(* Logix 5000 project; controller Kinematics_Delta_5D_with_Pick_n_Place 1756-L85E rev 33.11; software revision 33.00 *)

TASK MainTask (continuous, watchdog 500 ms) : MainProgram
TASK MotionEventTask (task) : VectorDynamics

MODULES
   Local : 1756-L85E (ICP 0, rev 33.11)
END_MODULES

TYPE SimOutputs :
STRUCT
   NumValues : DINT;   // Count of variables in the image
   D5_800_Y_ACT : REAL;   // Physics://physics/physics/D5-800/D5-800?_Y_ACT
   D5_800_Z_ACT : REAL;   // Physics://physics/physics/D5-800/D5-800?_Z_ACT
   D5_800_X_ACT : REAL;   // Physics://physics/physics/D5-800/D5-800?_X_ACT
   D5_800_R1_ACT : REAL;   // Physics://physics/physics/D5-800/D5-800?_R1_ACT
   D5_800_R2_ACT : REAL;   // Physics://physics/physics/D5-800/D5-800?_R2_ACT
   D5_800_GRIP : BOOL;   // Physics://physics/physics/D5-800/D5-800?_GRIP
END_STRUCT
END_TYPE

ADD_ON_INSTRUCTION deltaHomeArms   (* revision 1.0 *)

ROUTINE EnableInFalse   (* ladder *)
END_ROUTINE

ROUTINE Logic   (* ladder *)
END_ROUTINE
END_ADD_ON_INSTRUCTION

ADD_ON_INSTRUCTION Forward_Kinematics   (* revision 1.0, vendor Rockwell Automation *)
// This AOI will perform forward kinematics for Six axis articulated independent robot

ROUTINE Logic   (* structured text *)
   
END_ROUTINE
END_ADD_ON_INSTRUCTION

ADD_ON_INSTRUCTION homeToPositionError   (* revision 1.0, ExecuteEnableInFalse *)

ROUTINE EnableInFalse   (* ladder *)
END_ROUTINE

ROUTINE Logic   (* ladder *)
END_ROUTINE
END_ADD_ON_INSTRUCTION

ADD_ON_INSTRUCTION PICKPLACE   (* revision 1.0, ExecutePrescan *)
// Revision note:
// This AOI exhibits the PICK and PLACE behavior for a virtual cartesian axes.

ROUTINE Logic   (* ladder *)
END_ROUTINE

ROUTINE Prescan   (* ladder *)
// Move Step
END_ROUTINE
END_ADD_ON_INSTRUCTION

VAR_GLOBAL   (* controller tags *)
   a1_move_to_initialposition : BOOL;
   a2_mctTurnOn : BOOL;
   AccDec : REAL := 6666.665;
   Actual_Position_axis : REAL[3] := ([0] := 281.0, [2] := -1065.0219);
   AutoBrake : BOOL;
   Axis_Homing : BOOL;
   backOffAngle : REAL := 30.0;
   brakeAutoConstant : SINT; {constant}
   brakeReleaseConstant : SINT := 1; {constant}
   Cart_Vector_Speed_Sqr : REAL;
   Cart_Vector_Velocity_Sqr : REAL;
   CartSpeed : REAL := 500.0;
   CartVectorVelocity : REAL;
   CommandTolerance : REAL := 50.0;
   Counter : COUNTER := (PRE := 2, ACC := 1);
   CS_XYZRxRyRz : COORDINATE_SYSTEM;
   CycleTime : TIMER := (PRE := 99999, ACC := 99999, EN := 1, DN := 1);
   Delta5D_J1J2J3J4J5 : COORDINATE_SYSTEM;
   DeltaHomeArms : BOOL;
   DHA : deltaHomeArms;
   DownDist : REAL[3] := ([2] := -60.0);
   Downdistance : REAL := 80.0;
   DownDistBack : REAL := -120.0;
   dyn_data : DYNAMICS_DATA := (TimeUnits := 1, Profile := 1, Speed := 10.0, Acceleration := 5.0, Deceleration := 5.0, AccelerationJerk := 100.0, DecelerationJerk := 100.0, OrientationSpeed := 10.0, OrientationAcceleration := 30.0, OrientationDeceleration := 30.0);
   forAllAxes : BOOL;
   forArmsOnly : BOOL;
   forAxis1 : BOOL := 1;
   forAxis2 : BOOL := 1;
   forAxis3 : BOOL := 1;
   forAxis4 : BOOL;
   forAxis5 : BOOL;
   forNoAxes : BOOL;
   H2PE_1 : homeToPositionError;
   HalfHorizonMCLM : MOTION_INSTRUCTION := (FLAGS := -1442840576, EN := 1, DN := 1, PC := 1);
   homeMCPM : PATH_DATA[1] := ([0].InterpolationType := 1, [0].Position[0] := -20.012327, [0].Position[1] := 79.85217, [0].Position[2] := -7.858248, [0].Position[3] := -0.007234964, [0].Position[4] := 18.006336, [0].Position[5] := -20.005451, [0].RobotConfiguration := 6, [0].TerminationType := 1);
   HomePos : REAL[8] := ([0] := -20.012327, [1] := 79.85217, [2] := -7.858248, [3] := -0.007234964, [4] := 18.006336, [5] := -20.005451);
   HomeToTorque : BOOL;
   HorizDistance : REAL[3] := ([0] := -150.0);
   HorizDistBack : REAL := -360.0;
   HorizontalDistance : REAL := 360.0;
   InitialMclm1 : MOTION_INSTRUCTION;
   InitialPos : BOOL;
   Initiate_MCTO : BOOL;
   J1_Pos : REAL := 28.4;
   J1_v : AXIS_VIRTUAL;
   J2_Pos : REAL := 4.911;
   J2_v : AXIS_VIRTUAL;
   J3_Pos : REAL := -0.165;
   J3_v : AXIS_VIRTUAL;
   J4_Pos : REAL := -36.107;
   J4_v : AXIS_VIRTUAL;
   j4Angle : REAL := 180.0;
   j4AngleReturn : REAL := -180.0;
   J5_Pos : REAL := 35.032;
   J5_v : AXIS_VIRTUAL;
   j5Angle : REAL := 120.0;
   j5AngleReturn : REAL := -120.0;
   J6_Pos : REAL := -78.86052;
   J6_v : AXIS_VIRTUAL;
   junk1 : BOOL;
   LocalStep : DINT;
   LocalStep1 : DINT := 3;
   mah1 : MOTION_INSTRUCTION := (FLAGS := 704643072, DN := 1, PC := 1, STATE := 17);
   mah2 : MOTION_INSTRUCTION := (FLAGS := 704643072, DN := 1, PC := 1, STATE := 17);
   mah3 : MOTION_INSTRUCTION := (FLAGS := 704643072, DN := 1, PC := 1, STATE := 17);
   mah4 : MOTION_INSTRUCTION := (FLAGS := 704643072, DN := 1, PC := 1, STATE := 17);
   mah5 : MOTION_INSTRUCTION := (FLAGS := 704643072, DN := 1, PC := 1, STATE := 17);
   Mah_Ctr : MOTION_INSTRUCTION[10] := ([0].FLAGS := 33554432, [1].FLAGS := 33554432, [2].FLAGS := 33554432, [3].FLAGS := 33554432, [4].FLAGS := 33554432);
   maj1 : MOTION_INSTRUCTION := (FLAGS := 637534208, DN := 1, IP := 1);
   majMaster : REAL := 1.0;
   MAM_TO_ZERO : MOTION_INSTRUCTION[3] := ([0].FLAGS := 33554432, [1].FLAGS := 33554432, [2].FLAGS := 33554432);
   MAS : MOTION_INSTRUCTION[5] := ([0].FLAGS := 33554432, [1].FLAGS := 33554432, [2].FLAGS := 33554432, [3].FLAGS := 33554432, [4].FLAGS := 33554432);
   mas1 : MOTION_INSTRUCTION := (FLAGS := 33554432);
   masterZeroAngle : REAL := -82.04;
   MaxAccDec : REAL;
   MaxAccel : REAL := 70000.0;
   mccd1 : MOTION_INSTRUCTION;
   mccdOn : BOOL;
   mcpm : MOTION_INSTRUCTION[10] := ([0].FLAGS := 33554432, [1].FLAGS := 33554432, [2].FLAGS := 33554432, [3].FLAGS := 33554432, [4].FLAGS := 33554432, [5].FLAGS := 33554432, [6].FLAGS := 33554432, [7].FLAGS := 33554432, [8].FLAGS := 33554432);
   MCPM_Absolute_Move : BOOL;
   mcpm_ctr : MOTION_INSTRUCTION := (FLAGS := 33554432);
   MCPM_Incremental_Move : BOOL;
   mcpm_path : PATH_DATA[10] := ([0].InterpolationType := 1, [0].Position[0] := 100.0, [0].Position[1] := 200.0, [0].Position[2] := 300.0, [0].Position[3] := 30.0, [0].Position[4] := 20.0, [0].Position[5] := 10.0, [0].TerminationType := 1, [1].InterpolationType := 1, [1].Position[0] := 200.0, [1].Position[1] := 300.0, [1].Position[2] := 100.0, [1].Position[3] := 20.0, [1].Position[4] := 30.0, [1].Position[5] := 10.0, [1].TerminationType := 1, [2].InterpolationType := 1, [2].TerminationType := 1, [3].InterpolationType := 1, [3].Position[0] := 400.0, [3].Position[1] := 250.0, [3].Position[2] := 350.0, [3].Position[3] := 60.0, [3].Position[4] := 45.0, [3].Position[5] := 65.0);
   MCPM_RzMove_Coupling : BOOL;
   MCPM_with_WorkTool : BOOL;
   MCSOn : BOOL;
   mct1 : MOTION_INSTRUCTION := (FLAGS := 33554432);
   mctOn : BOOL := 1;
   mdcc1 : MOTION_INSTRUCTION := (FLAGS := 33554432);
   MotionAxisHome : BOOL;
   MotionAxisStop : BOOL;
   MotionServoOff : BOOL;
   MotionServoOn : BOOL;
   MoveArmsToZero : BOOL;
   MoveDown : BOOL;
   moveSpeed : REAL := 2.0;
   moveToZeroAccelAndJerk : REAL := 50.0;
   moveToZeroSpeed : REAL := 5.0;
   MSF : MOTION_INSTRUCTION[5] := ([0].FLAGS := 33554432, [1].FLAGS := 33554432, [2].FLAGS := 33554432, [3].FLAGS := 33554432, [4].FLAGS := 33554432);
   MSO : MOTION_INSTRUCTION[5] := ([0].FLAGS := 33554432, [1].FLAGS := 33554432, [2].FLAGS := 33554432, [3].FLAGS := 33554432, [4].FLAGS := 33554432);
   msoJ1 : MOTION_INSTRUCTION := (FLAGS := 33554432);
   msoJ2 : MOTION_INSTRUCTION := (FLAGS := 33554432);
   msoJ3 : MOTION_INSTRUCTION := (FLAGS := 33554432);
   msoJ4 : MOTION_INSTRUCTION := (FLAGS := 33554432);
   msoJ5 : MOTION_INSTRUCTION := (FLAGS := 33554432);
   OldCartSpeed : REAL;
   Ori_Vector_Speed_Sqr : REAL;
   Ori_Vector_Velocity_Sqr : REAL;
   ort : REAL[3];
   OrtVectorVelocity : REAL;
   path : PATH_DATA[10];
   PathPositions : REAL[8] := ([0] := 476.104, [1] := 2.682, [2] := -1200.037, [3] := 180.0);
   PathPositions1 : REAL[8] := ([0] := 498.811, [1] := -51.046, [2] := -885.044, [4] := -90.0, [5] := 135.0);
   PathPositions2 : REAL[8] := ([0] := -48.009, [1] := -19.226, [2] := -930.044, [3] := 180.0, [5] := -45.0);
   PathPositions3 : REAL[8] := ([0] := -145.893, [1] := 2.719, [2] := -1155.048, [4] := -90.0);
   PathPositions4 : REAL[8] := ([0] := 400.00003, [1] := 199.99995, [2] := 300.0, [3] := -179.99901, [4] := -0.0009865595, [5] := 90.0);
   PathPositions5 : REAL[8] := ([0] := 399.99997, [1] := -145.68004, [2] := 300.0, [3] := -179.999, [4] := -0.0010051423, [5] := 180.0);
   PathPositions6 : REAL[8] := ([0] := 399.99597, [1] := -145.68709, [2] := 7.3754336e-10, [3] := -179.99799, [4] := -0.0010051426, [5] := 180.0);
   pauseMove : DINT := 1;
   Pick_cycles_per_minute : REAL := 0.6000059;
   PickPlace2 : PICKPLACE;
   Place : BOOL;
   posArray : REAL[3] := ([0] := -180.0, [2] := -620.0);
   posErrThresh : REAL := 0.4;
   ReleaseBrake : BOOL;
   Robot : MOTION_GROUP;
   Rx : AXIS_VIRTUAL;
   Ry : AXIS_VIRTUAL;
   Rz : AXIS_VIRTUAL;
   simOutputs : SimOutputs := (NumValues := 6, D5_800_Z_ACT := -0.74696803, D5_800_X_ACT := 0.25423348, D5_800_R1_ACT := 1.2645825);
   SpeedOverwrite : BOOL;
   Start_AOI : BOOL;
   Start_MCPM : BOOL;
   Start_PickPlace : BOOL;
   step : DINT;
   Stop_Program : BOOL;
   T_CycleFrequency : REAL := 0.6000059;
   TermType1 : DINT := 1;
   test_1 : Forward_Kinematics;
   TimeinSeconds : REAL := 99.999;
   toolframe : POSITION_DATA;
   trs : REAL[3];
   turnsCtr : INT;
   unlatch : BOOL;
   UpDistance : REAL := 80.0;
   UpdistanceBack : REAL := -80.0;
   VectorAcceleration : REAL;
   VectorVelocity : REAL;
   VertDist : REAL := 80.0;
   VertDistance : REAL[3] := ([2] := -40.0);
   VerticalMCLM : MOTION_INSTRUCTION := (FLAGS := -1442840576, EN := 1, DN := 1, PC := 1);
   VirtualMaster : AXIS_VIRTUAL;
   workframe : POSITION_DATA;
   X : AXIS_VIRTUAL;
   X_Pos : REAL := 293.40237;
   Y : AXIS_VIRTUAL;
   Y_Pos : REAL;
   Z : AXIS_VIRTUAL;
   Z_Pos : REAL := 392.35858;
END_VAR

PROGRAM MainProgram   (* main routine a1_MainRoutine *)
VAR
   Autonox_Path : PATH_DATA[20] := ([0].InterpolationType := 1, [0].Position[0] := 281.0, [0].Position[2] := -1065.022, [0].Position[3] := 180.0, [0].TerminationType := 1, [0].CommandToleranceLinear := 200.0, [1].InterpolationType := 1, [1].Position[2] := 200.0, [1].MoveType := 1, [1].TerminationType := 6, [1].CommandToleranceLinear := 50.0, [2].InterpolationType := 1, [2].Position[0] := -400.0, [2].Position[4] := -45.0, [2].Position[5] := 45.0, [2].MoveType := 1, [2].TerminationType := 6, [2].CommandToleranceLinear := 50.0, [3].InterpolationType := 1, [3].Position[2] := -200.0, [3].Position[4] := -45.0, [3].Position[5] := 45.0, [3].MoveType := 1, [3].TerminationType := 6, [3].CommandToleranceLinear := 50.0, [4].InterpolationType := 1, [4].Position[1] := 300.0, [4].MoveType := 1, [4].TerminationType := 1, [4].CommandToleranceLinear := 50.0, [5].InterpolationType := 1, [5].Position[1] := -300.0, [5].MoveType := 1, [5].TerminationType := 6, [5].CommandToleranceLinear := 50.0, [6].InterpolationType := 1, [6].Position[2] := 200.0, [6].Position[4] := 45.0, [6].Position[5] := -45.0, [6].MoveType := 1, [6].TerminationType := 6, [6].CommandToleranceLinear := 50.0, [7].InterpolationType := 1, [7].Position[0] := 400.0, [7].Position[4] := 45.0, [7].Position[5] := -45.0, [7].MoveType := 1, [7].TerminationType := 6, [7].CommandToleranceLinear := 50.0, [8].InterpolationType := 1, [8].Position[2] := -200.0, [8].MoveType := 1, [8].TerminationType := 1, [8].CommandToleranceLinear := 50.0);
   Cartesian_Acceleration : REAL;
   Cartesian_Velocity : REAL;
   Codian_Abs_Rz_Path : PATH_DATA[20] := ([0].InterpolationType := 1, [0].Position[0] := 100.0, [0].Position[2] := -900.0, [0].Position[3] := 180.0, [0].TerminationType := 1, [0].CommandToleranceLinear := 200.0, [1].InterpolationType := 1, [1].Position[0] := 100.0, [1].Position[2] := -800.0, [1].Position[3] := 180.0, [1].TerminationType := 6, [1].CommandToleranceLinear := 50.0, [2].InterpolationType := 1, [2].Position[0] := -100.0, [2].Position[2] := -800.0, [2].Position[3] := 180.0, [2].Position[5] := 45.0, [2].TurnsCounters[1] := -2, [2].TerminationType := 6, [2].CommandToleranceLinear := 50.0, [3].InterpolationType := 1, [3].Position[0] := -100.0, [3].Position[2] := -900.0, [3].Position[3] := 180.0, [3].Position[5] := 90.0, [3].TurnsCounters[1] := -2, [3].TerminationType := 6, [3].CommandToleranceLinear := 50.0, [4].InterpolationType := 1, [4].Position[0] := -100.0, [4].Position[1] := 100.0, [4].Position[2] := -900.0, [4].Position[3] := 180.0, [4].Position[5] := 90.0, [4].TurnsCounters[1] := -2, [4].TerminationType := 1, [4].CommandToleranceLinear := 50.0, [5].InterpolationType := 1, [5].Position[0] := -100.0, [5].Position[2] := -900.0, [5].Position[3] := 180.0, [5].Position[5] := 90.0, [5].TurnsCounters[1] := -2, [5].TerminationType := 6, [5].CommandToleranceLinear := 50.0, [6].InterpolationType := 1, [6].Position[0] := -100.0, [6].Position[2] := -800.0, [6].Position[3] := 180.0, [6].Position[5] := 45.0, [6].TurnsCounters[1] := -2, [6].TerminationType := 6, [6].CommandToleranceLinear := 50.0, [7].InterpolationType := 1, [7].Position[0] := 100.0, [7].Position[2] := -800.0, [7].Position[3] := 180.0, [7].TerminationType := 6, [7].CommandToleranceLinear := 50.0, [8].InterpolationType := 1,
        [8].Position[0] := 100.0, [8].Position[2] := -900.0, [8].Position[3] := 180.0, [8].TerminationType := 1, [8].CommandToleranceLinear := 50.0);
   CUP : REAL := 0.003;
   Delta5D_Abs_Path : PATH_DATA[20] := ([0].InterpolationType := 1, [0].Position[0] := 100.0, [0].Position[2] := -900.0, [0].Position[3] := 180.0, [0].TerminationType := 1, [0].CommandToleranceLinear := 200.0, [1].InterpolationType := 1, [1].Position[0] := 100.0, [1].Position[2] := -800.0, [1].Position[3] := 180.0, [1].TerminationType := 6, [1].CommandToleranceLinear := 50.0, [2].InterpolationType := 1, [2].Position[0] := -100.0, [2].Position[2] := -800.0, [2].Position[3] := 180.0, [2].Position[4] := -45.0, [2].Position[5] := 45.0, [2].TurnsCounters[1] := -2, [2].TerminationType := 6, [2].CommandToleranceLinear := 50.0, [3].InterpolationType := 1, [3].Position[0] := -100.0, [3].Position[2] := -900.0, [3].Position[4] := -90.0, [3].Position[5] := -90.0, [3].TurnsCounters[1] := -2, [3].TerminationType := 6, [3].CommandToleranceLinear := 50.0, [4].InterpolationType := 1, [4].Position[0] := -100.0, [4].Position[1] := 100.0, [4].Position[2] := -900.0, [4].Position[4] := -90.0, [4].Position[5] := -90.0, [4].TurnsCounters[1] := -2, [4].TerminationType := 1, [4].CommandToleranceLinear := 50.0, [5].InterpolationType := 1, [5].Position[0] := -100.0, [5].Position[2] := -900.0, [5].Position[4] := -90.0, [5].Position[5] := -90.0, [5].TurnsCounters[1] := -2, [5].TerminationType := 6, [5].CommandToleranceLinear := 50.0, [6].InterpolationType := 1, [6].Position[0] := -100.0, [6].Position[2] := -800.0, [6].Position[3] := 180.0, [6].Position[4] := -45.0, [6].Position[5] := 45.0, [6].TurnsCounters[1] := -2, [6].TerminationType := 6, [6].CommandToleranceLinear := 50.0, [7].InterpolationType := 1, [7].Position[0] := 100.0, [7].Position[2] := -800.0, [7].Position[3] := 180.0, [7].TerminationType := 6,
        [7].CommandToleranceLinear := 50.0, [8].InterpolationType := 1, [8].Position[0] := 100.0, [8].Position[2] := -900.0, [8].Position[3] := 180.0, [8].TerminationType := 1, [8].CommandToleranceLinear := 50.0);
   Delta5D_Inc_Path : PATH_DATA[20] := ([0].InterpolationType := 1, [0].Position[0] := 100.0, [0].Position[2] := -900.0, [0].Position[3] := 180.0, [0].TerminationType := 1, [0].CommandToleranceLinear := 200.0, [1].InterpolationType := 1, [1].Position[2] := 100.0, [1].MoveType := 1, [1].TerminationType := 6, [1].CommandToleranceLinear := 50.0, [2].InterpolationType := 1, [2].Position[0] := -200.0, [2].Position[4] := -45.0, [2].Position[5] := 765.0, [2].MoveType := 1, [2].TerminationType := 6, [2].CommandToleranceLinear := 50.0, [3].InterpolationType := 1, [3].Position[2] := -100.0, [3].Position[4] := -45.0, [3].Position[5] := 45.0, [3].MoveType := 1, [3].TerminationType := 6, [3].CommandToleranceLinear := 50.0, [4].InterpolationType := 1, [4].Position[1] := 100.0, [4].MoveType := 1, [4].TerminationType := 1, [4].CommandToleranceLinear := 50.0, [5].InterpolationType := 1, [5].Position[1] := -100.0, [5].MoveType := 1, [5].TerminationType := 6, [5].CommandToleranceLinear := 50.0, [6].InterpolationType := 1, [6].Position[2] := 100.0, [6].Position[4] := 45.0, [6].Position[5] := -45.0, [6].MoveType := 1, [6].TerminationType := 6, [6].CommandToleranceLinear := 50.0, [7].InterpolationType := 1, [7].Position[0] := 200.0, [7].Position[4] := 45.0, [7].Position[5] := -765.0, [7].MoveType := 1, [7].TerminationType := 6, [7].CommandToleranceLinear := 50.0, [8].InterpolationType := 1, [8].Position[2] := -100.0, [8].MoveType := 1, [8].TerminationType := 1, [8].CommandToleranceLinear := 50.0);
   Delta5D_Path : PATH_DATA[20] := ([0].InterpolationType := 1, [0].Position[0] := 100.0, [0].Position[2] := -900.0, [0].Position[3] := 180.0, [0].TerminationType := 1, [0].CommandToleranceLinear := 200.0, [1].InterpolationType := 1, [1].Position[2] := 100.0, [1].MoveType := 1, [1].TerminationType := 6, [1].CommandToleranceLinear := 50.0, [2].InterpolationType := 1, [2].Position[0] := -200.0, [2].Position[4] := -45.0, [2].Position[5] := 765.0, [2].MoveType := 1, [2].TerminationType := 6, [2].CommandToleranceLinear := 50.0, [3].InterpolationType := 1, [3].Position[2] := -100.0, [3].Position[4] := -45.0, [3].Position[5] := 45.0, [3].MoveType := 1, [3].TerminationType := 6, [3].CommandToleranceLinear := 50.0, [4].InterpolationType := 1, [4].Position[1] := 100.0, [4].MoveType := 1, [4].TerminationType := 1, [4].CommandToleranceLinear := 50.0, [5].InterpolationType := 1, [5].Position[1] := -100.0, [5].MoveType := 1, [5].TerminationType := 6, [5].CommandToleranceLinear := 50.0, [6].InterpolationType := 1, [6].Position[2] := 100.0, [6].Position[4] := 45.0, [6].Position[5] := -45.0, [6].MoveType := 1, [6].TerminationType := 6, [6].CommandToleranceLinear := 50.0, [7].InterpolationType := 1, [7].Position[0] := 200.0, [7].Position[4] := 45.0, [7].Position[5] := -765.0, [7].MoveType := 1, [7].TerminationType := 6, [7].CommandToleranceLinear := 50.0, [8].InterpolationType := 1, [8].Position[2] := -100.0, [8].MoveType := 1, [8].TerminationType := 1, [8].CommandToleranceLinear := 50.0);
   Delta5D_Work_Tool_Path : PATH_DATA[20] := ([0].InterpolationType := 1, [0].Position[3] := 180.0, [0].TerminationType := 1, [0].CommandToleranceLinear := 200.0, [1].InterpolationType := 1, [1].Position[2] := 100.0, [1].MoveType := 1, [1].TerminationType := 6, [1].CommandToleranceLinear := 50.0, [2].InterpolationType := 1, [2].Position[0] := -200.0, [2].Position[4] := -45.0, [2].Position[5] := 765.0, [2].MoveType := 1, [2].TerminationType := 6, [2].CommandToleranceLinear := 50.0, [3].InterpolationType := 1, [3].Position[2] := -100.0, [3].Position[4] := -45.0, [3].Position[5] := 45.0, [3].MoveType := 1, [3].TerminationType := 6, [3].CommandToleranceLinear := 50.0, [4].InterpolationType := 1, [4].Position[1] := 100.0, [4].MoveType := 1, [4].TerminationType := 1, [4].CommandToleranceLinear := 50.0, [5].InterpolationType := 1, [5].Position[1] := -100.0, [5].MoveType := 1, [5].TerminationType := 6, [5].CommandToleranceLinear := 50.0, [6].InterpolationType := 1, [6].Position[2] := 100.0, [6].Position[4] := 45.0, [6].Position[5] := -45.0, [6].MoveType := 1, [6].TerminationType := 6, [6].CommandToleranceLinear := 50.0, [7].InterpolationType := 1, [7].Position[0] := 200.0, [7].Position[4] := 45.0, [7].Position[5] := -765.0, [7].MoveType := 1, [7].TerminationType := 6, [7].CommandToleranceLinear := 50.0, [8].InterpolationType := 1, [8].Position[2] := -100.0, [8].MoveType := 1, [8].TerminationType := 1, [8].CommandToleranceLinear := 50.0);
   dyndata : DYNAMICS_DATA := (TimeUnits := 1, Profile := 1, Speed := 100.0, Acceleration := 100.0, Deceleration := 100.0, AccelerationJerk := 100.0, DecelerationJerk := 100.0, OrientationSpeed := 100.0, OrientationAcceleration := 100.0, OrientationDeceleration := 100.0);
   initalPath : PATH_DATA[1] := ([0].InterpolationType := 1, [0].TerminationType := 1);
   MASAll : BOOL;
   mcpm1 : MOTION_INSTRUCTION := (FLAGS := 33554432);
   MCPM_ToolFrame : POSITION_DATA;
   MCPM_WorkFrame : POSITION_DATA := (X := 27.5, Z := -781.968);
   mcs1 : MOTION_INSTRUCTION := (FLAGS := 33554432);
   mcs2 : MOTION_INSTRUCTION := (FLAGS := 33554432);
   MCSCart : BOOL;
   MCSRobot : BOOL;
   mcto1 : MOTION_INSTRUCTION := (FLAGS := 33554432);
   old_cartesian_average_Velocity : REAL;
   pauseMSO : BOOL;
   pauseTransforms : BOOL;
   PickPlace1 : PICKPLACE;
   StartTransforms : BOOL;
   StartTransforms1 : BOOL;
END_VAR

ROUTINE a1_MainRoutine   (* ladder *)
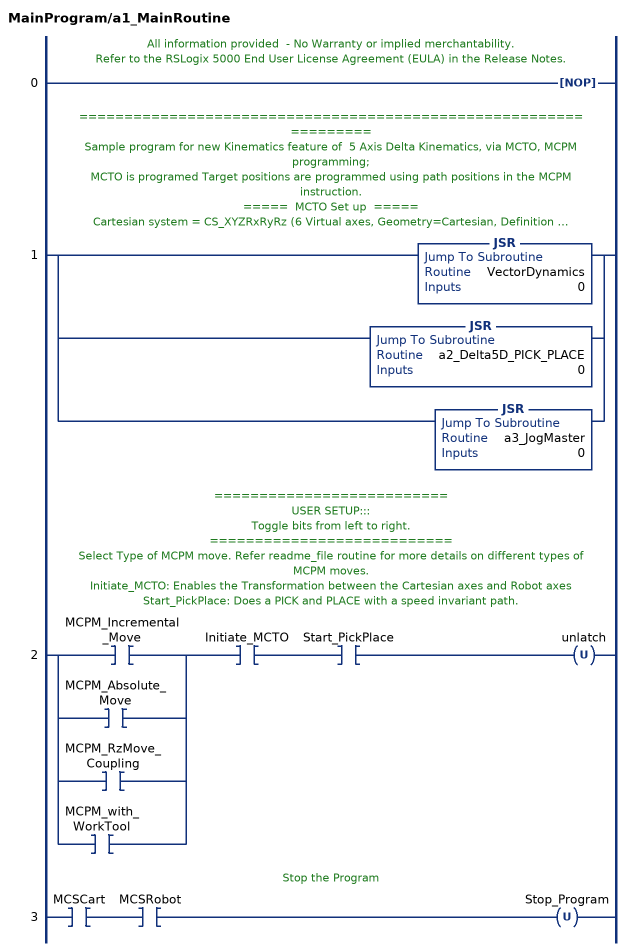
   // All information provided  - No Warranty or implied merchantability.
   // Refer to the RSLogix 5000 End User License Agreement (EULA) in the Release Notes.
   0: NOP();
   // =================================================================
   // Sample program for new Kinematics feature of  5 Axis Delta Kinematics, via MCTO, MCPM programming;
   // MCTO is programed Target positions are programmed using path positions in the MCPM instruction.
   // =====  MCTO Set up  =====
   // Cartesian system = CS_XYZRxRyRz (6 Virtual axes, Geometry=Cartesian, Definition = XYZRxRyRz)
   // Robot coordinate system = Delta5D_J1J2J3J4J5 (5 Joint axes, Geometry=Delta 3D, Definition = J1J2J3J4J5)
   // ================================================================
   // Open Trend = to view the plot of robot’s TCP Positions
   // 	XY Plot shows object positions on the conveyor at TCP and End of Arm(EOA)
   // XZ Plot shows TCP moves during different pick cycles
   // ==================================================================
   1: [JSR(VectorDynamics,0) ,JSR(a2_Delta5D_PICK_PLACE,0) ,JSR(a3_JogMaster,0) ];
   // ==========================
   // USER SETUP:::
   // Toggle bits from left to right.
   // ===========================
   // Select Type of MCPM move. Refer readme_file routine for more details on different types of MCPM moves.
   //  Initiate_MCTO: Enables the Transformation between the Cartesian axes and Robot axes
   // Start_PickPlace: Does a PICK and PLACE with a speed invariant path.
   2: [XIC(MCPM_Incremental_Move) ,XIC(MCPM_Absolute_Move) ,XIC(MCPM_RzMove_Coupling) ,XIC(MCPM_with_WorkTool) ]XIC(Initiate_MCTO)XIC(Start_PickPlace)OTU(unlatch);
   // Stop the Program
   3: XIC(MCSCart)XIC(MCSRobot)OTU(Stop_Program);
END_ROUTINE

ROUTINE a2_Delta5D_PICK_PLACE   (* ladder *)
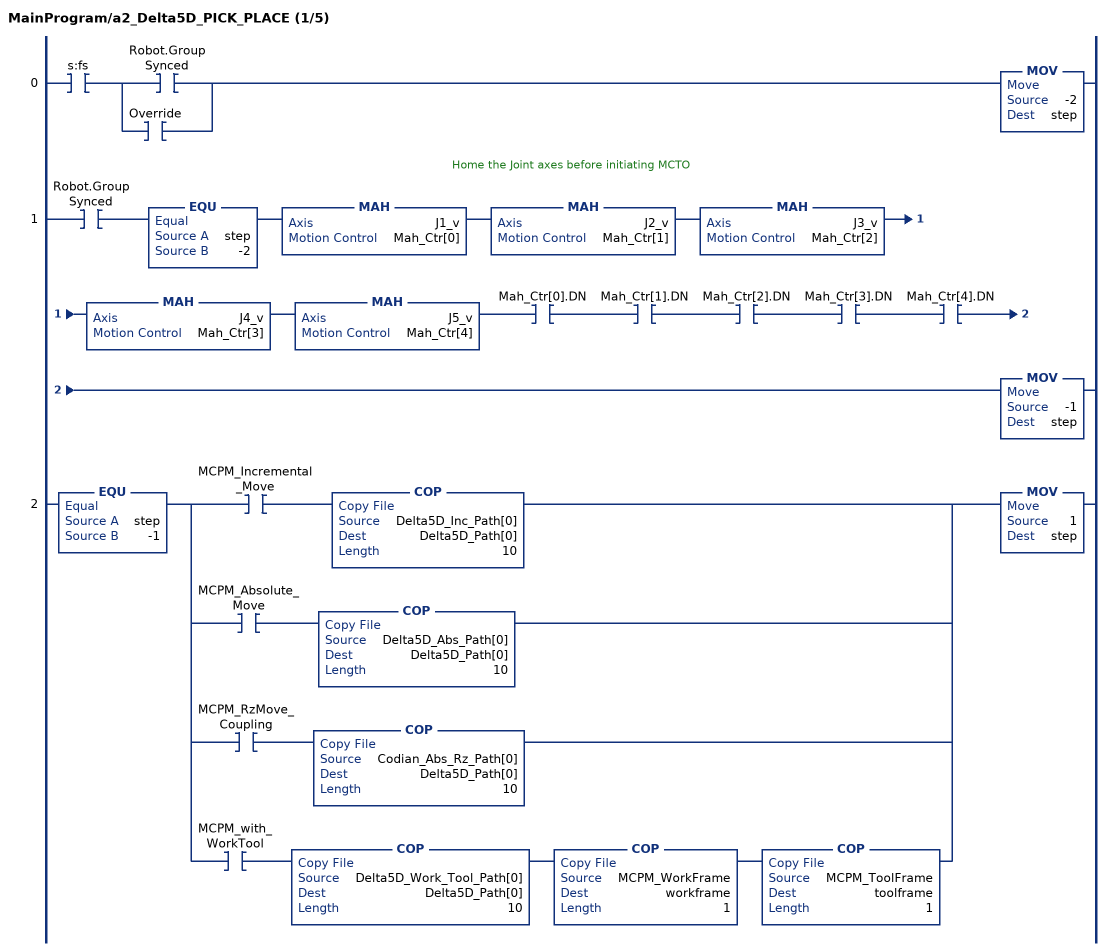
   0: XIC(s:fs)[XIC(Robot.GroupSynced) ,XIC(Override) ]MOV(-2,step);
   // Home the Joint axes before initiating MCTO
   1: XIC(Robot.GroupSynced)EQU(step,-2)MAH(J1_v,Mah_Ctr[0])MAH(J2_v,Mah_Ctr[1])MAH(J3_v,Mah_Ctr[2])MAH(J4_v,Mah_Ctr[3])MAH(J5_v,Mah_Ctr[4])XIC(Mah_Ctr[0].DN)XIC(Mah_Ctr[1].DN)XIC(Mah_Ctr[2].DN)XIC(Mah_Ctr[3].DN)XIC(Mah_Ctr[4].DN)MOV(-1,step);
   2: EQU(step,-1)[XIC(MCPM_Incremental_Move) COP(Delta5D_Inc_Path[0],Delta5D_Path[0],10) ,XIC(MCPM_Absolute_Move) COP(Delta5D_Abs_Path[0],Delta5D_Path[0],10) ,XIC(MCPM_RzMove_Coupling) COP(Codian_Abs_Rz_Path[0],Delta5D_Path[0],10) ,XIC(MCPM_with_WorkTool) COP(Delta5D_Work_Tool_Path[0],Delta5D_Path[0],10) COP(MCPM_WorkFrame,workframe,1) COP(MCPM_ToolFrame,toolframe,1) ]MOV(1,step);
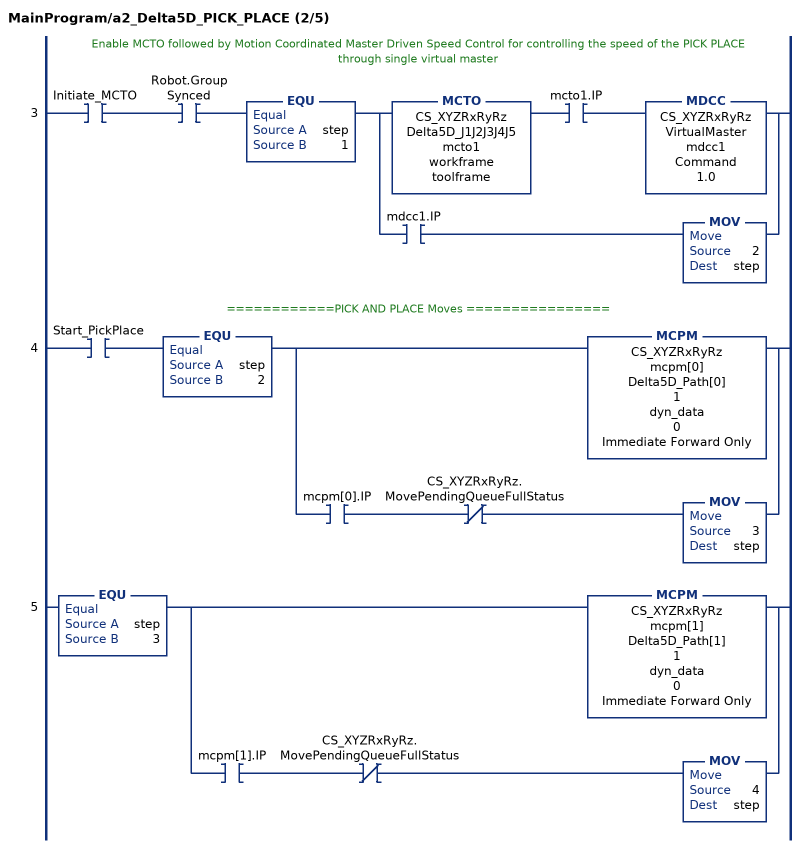
   // Enable MCTO followed by Motion Coordinated Master Driven Speed Control for controlling the speed of the PICK PLACE through single virtual master
   3: XIC(Initiate_MCTO)XIC(Robot.GroupSynced)EQU(step,1)[MCTO(CS_XYZRxRyRz,Delta5D_J1J2J3J4J5,mcto1,workframe,toolframe) XIC(mcto1.IP) MDCC(CS_XYZRxRyRz,VirtualMaster,mdcc1,Command,1.0) ,XIC(mdcc1.IP) MOV(2,step) ];
   // ============PICK AND PLACE Moves ================
   4: XIC(Start_PickPlace)EQU(step,2)[MCPM(CS_XYZRxRyRz,mcpm[0],Delta5D_Path[0],1,dyn_data,0,Immediate Forward Only) ,XIC(mcpm[0].IP) XIO(CS_XYZRxRyRz.MovePendingQueueFullStatus) MOV(3,step) ];
   5: EQU(step,3)[MCPM(CS_XYZRxRyRz,mcpm[1],Delta5D_Path[1],1,dyn_data,0,Immediate Forward Only) ,XIC(mcpm[1].IP) XIO(CS_XYZRxRyRz.MovePendingQueueFullStatus) MOV(4,step) ];
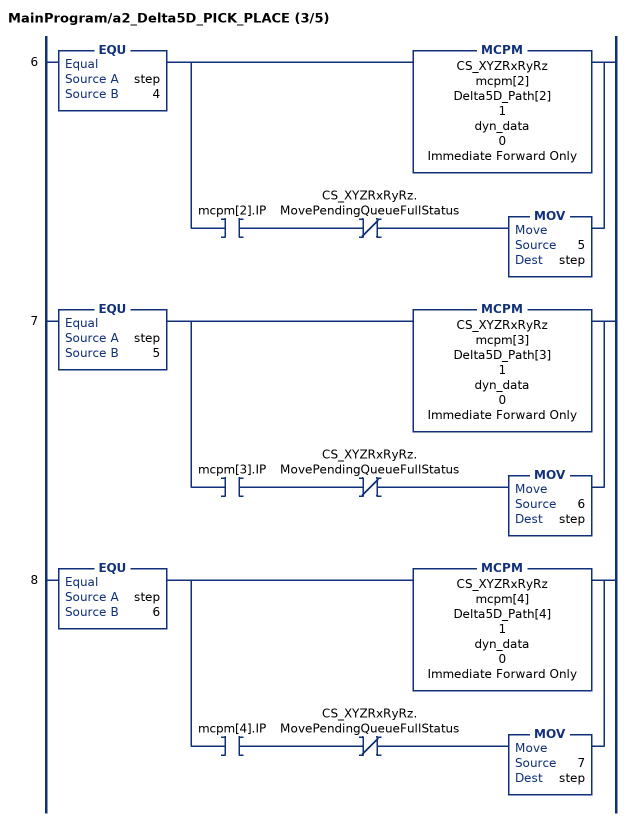
   6: EQU(step,4)[MCPM(CS_XYZRxRyRz,mcpm[2],Delta5D_Path[2],1,dyn_data,0,Immediate Forward Only) ,XIC(mcpm[2].IP) XIO(CS_XYZRxRyRz.MovePendingQueueFullStatus) MOV(5,step) ];
   7: EQU(step,5)[MCPM(CS_XYZRxRyRz,mcpm[3],Delta5D_Path[3],1,dyn_data,0,Immediate Forward Only) ,XIC(mcpm[3].IP) XIO(CS_XYZRxRyRz.MovePendingQueueFullStatus) MOV(6,step) ];
   8: EQU(step,6)[MCPM(CS_XYZRxRyRz,mcpm[4],Delta5D_Path[4],1,dyn_data,0,Immediate Forward Only) ,XIC(mcpm[4].IP) XIO(CS_XYZRxRyRz.MovePendingQueueFullStatus) MOV(7,step) ];
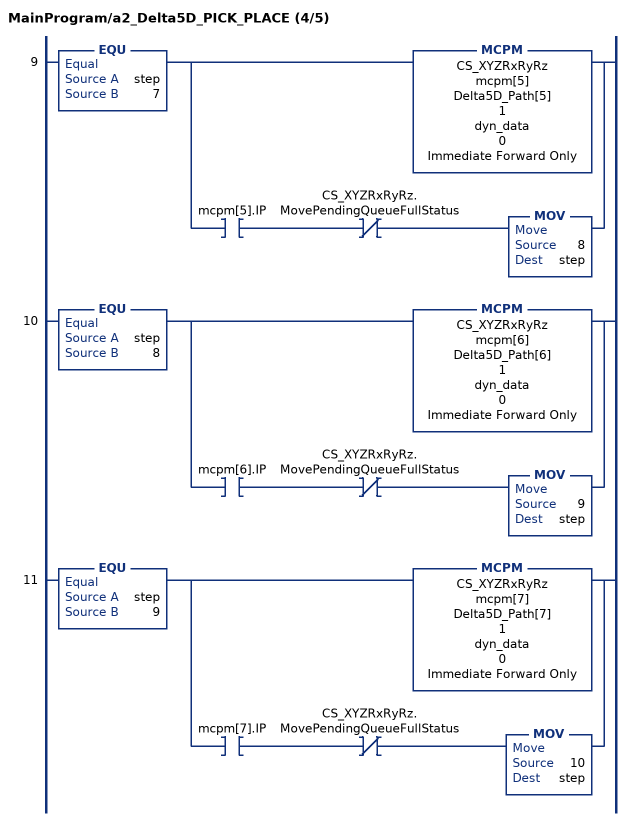
   9: EQU(step,7)[MCPM(CS_XYZRxRyRz,mcpm[5],Delta5D_Path[5],1,dyn_data,0,Immediate Forward Only) ,XIC(mcpm[5].IP) XIO(CS_XYZRxRyRz.MovePendingQueueFullStatus) MOV(8,step) ];
   10: EQU(step,8)[MCPM(CS_XYZRxRyRz,mcpm[6],Delta5D_Path[6],1,dyn_data,0,Immediate Forward Only) ,XIC(mcpm[6].IP) XIO(CS_XYZRxRyRz.MovePendingQueueFullStatus) MOV(9,step) ];
   11: EQU(step,9)[MCPM(CS_XYZRxRyRz,mcpm[7],Delta5D_Path[7],1,dyn_data,0,Immediate Forward Only) ,XIC(mcpm[7].IP) XIO(CS_XYZRxRyRz.MovePendingQueueFullStatus) MOV(10,step) ];
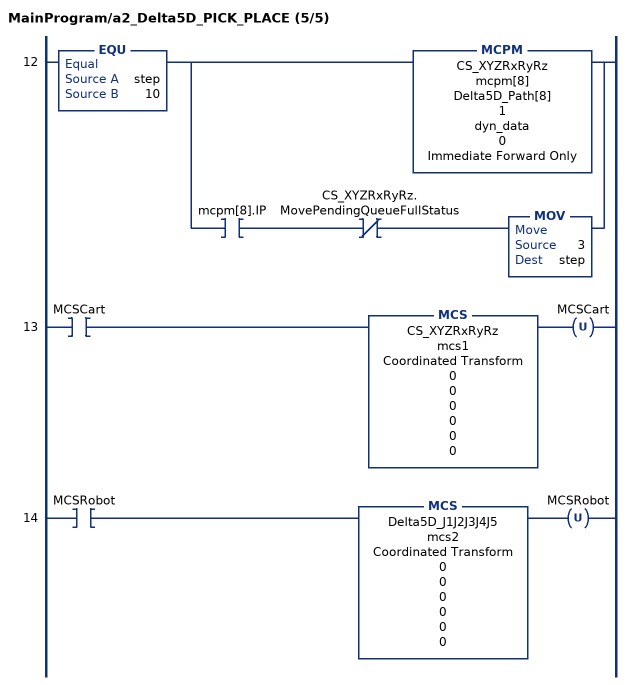
   12: EQU(step,10)[MCPM(CS_XYZRxRyRz,mcpm[8],Delta5D_Path[8],1,dyn_data,0,Immediate Forward Only) ,XIC(mcpm[8].IP) XIO(CS_XYZRxRyRz.MovePendingQueueFullStatus) MOV(3,step) ];
   13: XIC(MCSCart)MCS(CS_XYZRxRyRz,mcs1,Coordinated Transform,0,0,0,0,0,0)OTU(MCSCart);
   14: XIC(MCSRobot)MCS(Delta5D_J1J2J3J4J5,mcs2,Coordinated Transform,0,0,0,0,0,0)OTU(MCSRobot);
END_ROUTINE

ROUTINE a3_JogMaster   (* ladder *)
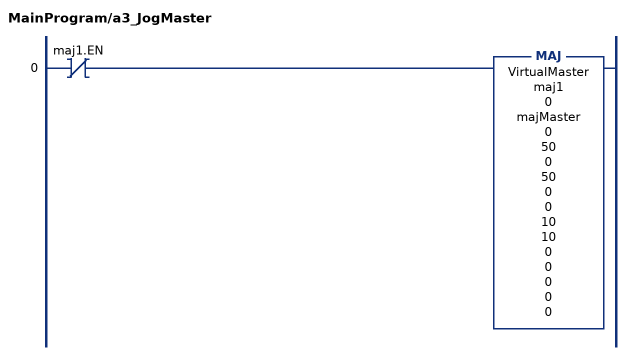
   0: XIO(maj1.EN)MAJ(VirtualMaster,maj1,0,majMaster,0,50,0,50,0,0,10,10,0,0,0,0,0);
END_ROUTINE

ROUTINE readme_file   (* structured text *)
   
   (*
    /*  ============================================================================= */
   				  DELTA 5 Axis Robot with Orientation Control
    /*  ============================================================================= */
   
   This program contains a 5-Axis Delta Robot demonstrating a simple PICK and PLACE in XYZ plane with Ry andRz orientation control.
   It also demonstrates the Speed override functionality (scaling the entire PICK and PLACE dynamics using a single master axis).
   
   
   a2_Delta5D_PICK_PLACE routine overview:
   
   1. MCTO links the Cartesian XYZRxRyRz and Delta-4Axis Robot Coordinate systems (Coordinate Definition for Delta 4 Axis is J1J2J3J6) and transforms the motion
   2. MDCC is the master driven speed control instruction that links the Cartesian coordinate system to the virtual master axis for speed override functionality.
   3. Using MCPM Path move instruction, the Robot is programmed to move to a known Absolute Start Position.
   4. Rest of the pick and place moves are programed different ways
   	a.	Incremental moves with Ry and Rz orientations
   
   	Incremental moves are programed with 100 Up (AB) followed by 400 horizontal (BC) and 100 down (CD)in XZ plane, last 100 (DE) on DE plane.
   	The same is repeated in the reverse direction for the PLACE move in YZ plane.
   	Along with the Cartesian moves, the Path moves are also programmed with Rz orientation.
   
   					 __________________________
   				  B |            400           | C
   				100 |                          |
   					|                          |100
   					|                          |      100
   				  A |                        D |__ __ __ __ E
   
   
   	 The Ry and Rz Orientation moves are programmed incremental along with the primary cartesian axes as below:
   		AB =   Ry@ 0  degrees and Rx@ 0    degrees
   		BC =   Ry@-45 degrees and Rx@ 765  degrees
   		CD =   Ry@-45 degrees and Rx@ 45   degrees
   		DE =   Ry@ 0  degrees and Rx@ 0    degrees
   		ED =   Ry@ 0  degrees and Rx@ 0    degrees
   		DC =   Ry@ 45 degrees and Rx@ -45  degrees
   		CB =   Ry@ 45 degrees and Rx@ -765 degrees
   		BA =   Ry@ 0  degrees and Rx@ 0    degrees
   
   
   	b.	Absolute moves with Ry and Rz orientations
   
   		Same A,B,C,D,E  Positions  shown are programmed using absolute positions.
   		Refer Delta5D_Abs_Path[].Position[] array for absolute position values.
   		Turns counter feature on J4 axis is used here for Rz moves.
   
   	c.	Absolute moves with only Rz orientations.
   
   		These moves will show specific “ J4:J5 coupling ration”feature of 5 axis Delta geometries.
   		When  you move only Rz axis it will move J4 and J5 axis to remove the coupling effect by J4 axis.
   		Rz positions are programmed using multiple turns with “Turns counter “feature.
   		Refer Delta5D_Abs_Rz_Path[].Position[] array for absolute position values.
   
   
   	d.	Incremental move with Work and Tool frame offsets.
   
   		These moves will show Work frame feature on 5 axis delta robots.
   		Work frame is transferred to End Of Arm of robot using work frame offset values.
   		Sometimes this will helps user to program target end position from EOA.
   		Work Frame offsets =  X= 27.5, Y = 0, Z = -781.968, Rx = 0 ,Ry = 0, Rz =0, Refer MCPM_WorkFrame parameter for Work frame offset values.
   		Refer Delta5D_Work_Tool_Path[].Position array for incremental end positions.
   
   6. The command tolerance for the first move is set to 100 units and the second move is set to 50  units for the PICK cycle.
   
   7. The dynamics of the path move are all programmed in % of max (dyn_data.UnitsMode  is set to 0).
   
   
   a3_JogMaster routine overview:
   1.	Jogging the VirtualMaster axis using MAJ instruction will provide the speed override functionality for the PICK and PLACE cycle.
   
   VectorDynamics. MainRoutine Overview:
   1. The routine calculates the Cartesian Vector velocity and the Orientation vector velocity.
   
   See online help 'Configure the Delta J1J2J3J4J5 Coordinate System' for more information on configuring Delta 5 axis Delta robots.
   See  online help 'Blending Path Moves with MCPM for more information on the PICK and PLACE Cycle'
   *)
   
END_ROUTINE

ROUTINE VectorDynamics   (* ladder *)
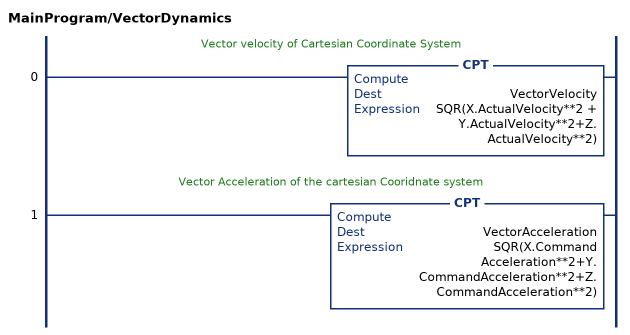
   // Vector velocity of Cartesian Coordinate System
   0: CPT(VectorVelocity,SQR(X.ActualVelocity**2 + Y.ActualVelocity**2+Z.ActualVelocity**2));
   // Vector Acceleration of the cartesian Cooridnate system
   1: CPT(VectorAcceleration,SQR(X.CommandAcceleration**2+Y.CommandAcceleration**2+Z.CommandAcceleration**2));
END_ROUTINE
END_PROGRAM

PROGRAM VectorDynamics   (* main routine eventTask *)

ROUTINE eventTask   (* ladder *)
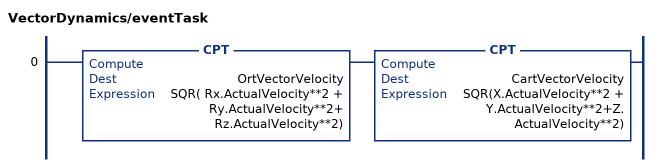
   0: CPT(OrtVectorVelocity,SQR( Rx.ActualVelocity**2 + Ry.ActualVelocity**2+ Rz.ActualVelocity**2))CPT(CartVectorVelocity,SQR(X.ActualVelocity**2 + Y.ActualVelocity**2+Z.ActualVelocity**2));
END_ROUTINE
END_PROGRAM
